% RSLogix 500 project I2P JOB5_BAK017.RSS, saved by version 10.00.00.00 %
PROJECT "UNTITLED"    % processor: Bul.1763 MicroLogix 1100 Series B %

PROGRAM FILES
  LAD 2   5 rungs

DATA FILES
  O0 OUTPUT  4 elements
  I1 INPUT  6 elements
  S2 STATUS  66 elements
  B3 BINARY  1 elements
  T4 TIMER  1 elements
  C5 COUNTER  1 elements
  R6 CONTROL  1 elements
  N7 INTEGER  1 elements
  F8 FLOAT  1 elements

LADDER 2
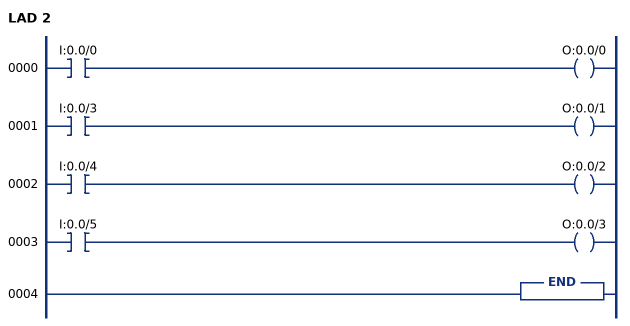
% Rung: 0 %
SOR XIC I:0.0/0 OTE O:0.0/0 EOR
% Rung: 1 %
SOR XIC I:0.0/3 OTE O:0.0/1 EOR
% Rung: 2 %
SOR XIC I:0.0/4 OTE O:0.0/2 EOR
% Rung: 3 %
SOR XIC I:0.0/5 OTE O:0.0/3 EOR
% Rung: 4 %
SOR END EOR
